# EPICS autosave request: iocBoot/ioc13Aerotech/auto_settings.req
file "CARS_motor_settings.req",         P=$(P), M=m1
